PROGRAM MAIN
VAR
END_VAR

PB_TestRunner();

END_PROGRAM

(* stored: Version 1.1.0.1, ProductVersion 3.1.4024.4
   POU MAIN: Id {a2561576-7611-4adb-8bbe-d412e59b6418}, SpecialFunc None *)
